FUNCTION_BLOCK PumpControl01
VAR_INPUT
	LsLow							:	BOOL;		// limit switch LOW (NO)
	LsMiddle						:	BOOL;		// limit switch MIDDLE (NO)
	LsHigh							:	BOOL;		// limit switch HIGH (NC)
END_VAR
VAR_OUTPUT
	Motor1							:	BOOL;		// motor 1 output
	Motor2							:	BOOL;		// motor 2 output
END_VAR
VAR
	AlternatePump					:	BOOL;		// flag for pump alternation
	RunMotor						:	BOOL;		// pump alternation control
END_VAR
VAR // added by the converter: edge detectors and wires of the graphical bodies
    _w1, _w2, _w3 : BOOL;
END_VAR

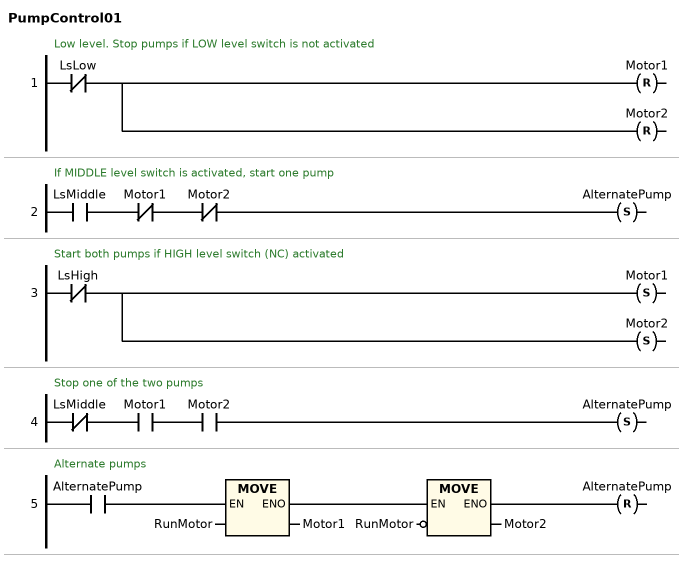
// NETWORK 1
// Low level. Stop pumps if LOW level switch is not activated
_w1 := NOT LsLow;
Motor1 R= _w1;
Motor2 R= _w1;

// NETWORK 2
// If MIDDLE level switch is activated, start one pump
AlternatePump S= LsMiddle AND NOT Motor1 AND NOT Motor2;

// NETWORK 3
// Start both pumps if HIGH level switch (NC) activated
_w2 := NOT LsHigh;
Motor1 S= _w2;
Motor2 S= _w2;

// NETWORK 4
// Stop one of the two pumps
AlternatePump S= NOT LsMiddle AND Motor1 AND Motor2;

// NETWORK 5
// Alternate pumps
_w3 := AlternatePump;
IF _w3 THEN Motor1 := RunMotor; END_IF
IF _w3 THEN Motor2 := NOT RunMotor; END_IF
AlternatePump R= _w3;

END_FUNCTION_BLOCK

(* stored: Version 1.1.0.1, ProductVersion 3.1.4024.15
   POU PumpControl01: Id {01e0fbed-ee07-403e-a377-86f0dbaf4cad}, SpecialFunc None *)
